FUNCTION_BLOCK IN_PRESS_BUTTON (* Button generating event when pressed and when released *)
  (* Standard: 61499-2 *)
  (* Version 1.0, 2006-01-02, Anirudha, UoA *)
  (* Compiler header: package fb.rt.student; *)
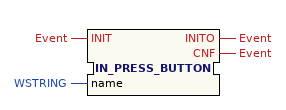
  EVENT_INPUT
    INIT; (* Initialization Request *)
  END_EVENT
  EVENT_OUTPUT
    INITO; (* Initialization Confirm *)
    CNF; (* Execution Confirmation *)
  END_EVENT
  VAR_INPUT
    name : WSTRING;
  END_VAR
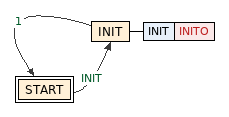
  EC_STATES
    START; (* Initial State *)
    INIT : INIT -> INITO; (* Initialization *)
  END_STATES
  EC_TRANSITIONS
    START TO INIT := INIT;
    INIT TO START := 1;
  END_TRANSITIONS
  ALGORITHM INIT IN ST: (* Initialization algorithm *)

  END_ALGORITHM
END_FUNCTION_BLOCK
